FUNCTION_BLOCK EL3164
VAR
	_io : EL3xx4_Data;
	{attribute addProperty Name "WcState"}
	_wcState : WcStateInputToggle;
	{attribute addProperty Name "Info data"}
	_infoData : InfoDataAds;
END_VAR

PROPERTY IO : REFERENCE TO EL3xx4_Data
GET
IO REF= _io;
END_GET
END_PROPERTY

PROPERTY WcState : REFERENCE TO WcStateInputToggle
GET
WcState REF= _wcState;
END_GET
END_PROPERTY

END_FUNCTION_BLOCK

(* stored: Version 1.1.0.1, ProductVersion 3.1.4024.9
   POU EL3164: Id {eec55c44-887b-0abc-2d86-879ed115b505}, SpecialFunc None
   Property IO: Id {998b9f71-ae78-03ae-38cb-c6ae46ef2897}
   Get Get: Id {24fc9212-08e8-0f3b-1cf6-3ad5154b2df1}
   Property WcState: Id {f394d82e-423a-0262-2a32-a8e1b8e04398}
   Get Get: Id {60e481f9-7e71-044f-1eb0-061200d84762} *)
